% RSLogix 500 project LINL0619_042121 download.RSS, saved by version 11.00.00.00 %
PROJECT "LINL0619"    % processor: MicroLogix 1400 %

PROGRAM FILES
  LAD 2   65 rungs
  LAD 3   9 rungs
  LAD 4   18 rungs
  LAD 5   11 rungs
  LAD 6   13 rungs
  LAD 7   5 rungs
  LAD 8   5 rungs
  LAD 9   26 rungs
  LAD 10   5 rungs
  LAD 11   6 rungs
  LAD 12   3 rungs
  LAD 13   7 rungs
  LAD 14   7 rungs
  LAD 81   21 rungs
  LAD 82   8 rungs
  LAD 83   6 rungs
  LAD 84   4 rungs
  LAD 85   9 rungs
  LAD 86   5 rungs
  LAD 87   5 rungs
  LAD 90   3 rungs
  LAD 91   9 rungs
  LAD 92   5 rungs
  LAD 93   3 rungs
  LAD 94   21 rungs
  LAD 95   7 rungs
  LAD 96   6 rungs
  LAD 97   4 rungs
  LAD 98   8 rungs
  LAD 99   5 rungs
  LAD 100   5 rungs
  LAD 101   7 rungs
  LAD 102   8 rungs
  LAD 103   3 rungs
  LAD 104   9 rungs
  LAD 105   7 rungs
  LAD 106   3 rungs
  LAD 135   3 rungs
  LAD 137   15 rungs
  LAD 138   13 rungs
  LAD 139   19 rungs
  LAD 140   8 rungs
  LAD 141   6 rungs
  LAD 142   6 rungs
  LAD 143   7 rungs
  LAD 144   8 rungs
  LAD 148   21 rungs
  LAD 149   7 rungs
  LAD 150   6 rungs
  LAD 151   4 rungs
  LAD 152   9 rungs
  LAD 153   5 rungs
  LAD 154   5 rungs
  LAD 155   10 rungs
  LAD 156   8 rungs
  LAD 157   3 rungs
  LAD 158   9 rungs
  LAD 159   5 rungs
  LAD 160   3 rungs
  LAD 161   21 rungs
  LAD 162   7 rungs
  LAD 163   5 rungs
  LAD 164   3 rungs
  LAD 165   8 rungs
  LAD 166   5 rungs
  LAD 167   5 rungs
  LAD 168   9 rungs
  LAD 169   8 rungs
  LAD 170   3 rungs
  LAD 171   9 rungs
  LAD 172   5 rungs
  LAD 173   3 rungs
  LAD 174   22 rungs
  LAD 175   7 rungs
  LAD 176   6 rungs
  LAD 177   4 rungs
  LAD 178   9 rungs
  LAD 179   5 rungs
  LAD 180   5 rungs
  LAD 181   9 rungs
  LAD 182   8 rungs
  LAD 183   3 rungs
  LAD 184   9 rungs
  LAD 185   5 rungs
  LAD 186   3 rungs
  LAD 187   22 rungs
  LAD 188   7 rungs
  LAD 189   6 rungs
  LAD 190   4 rungs
  LAD 191   9 rungs
  LAD 192   5 rungs
  LAD 193   5 rungs
  LAD 194   9 rungs
  LAD 195   8 rungs
  LAD 196   3 rungs
  LAD 197   9 rungs
  LAD 198   5 rungs
  LAD 199   3 rungs
  LAD 200   16 rungs
  LAD 235   7 rungs
  LAD 236   5 rungs
  LAD 237   4 rungs
  LAD 238   4 rungs
  LAD 239   4 rungs
  LAD 240   4 rungs
  LAD 241   4 rungs
  LAD 242   4 rungs
  LAD 243   4 rungs
  LAD 244   31 rungs
  LAD 245   8 rungs
  LAD 246   9 rungs
  LAD 247   6 rungs
  LAD 248   6 rungs
  LAD 249   8 rungs
  LAD 250   8 rungs
  LAD 251   8 rungs
  LAD 252   7 rungs
  LAD 253   7 rungs
  LAD 254   4 rungs
  LAD 255   18 rungs
  LAD 88, 89, 107, 108, 109, 110, 111, 112, 113, 114, 115, 116, 117, 118, 119, 120, 121, 122, 123, 124, 125, 126, 127, 128, 129, 130, 131, 132: only END

DATA FILES
  O0 OUTPUT  11 elements
  I1 INPUT  11 elements
  S2 STATUS  66 elements
  B3 BINARY  256 elements
  T4 TIMER  45 elements
  C5 COUNTER  1 elements
  R6 CONTROL  30 elements
  N7 INTEGER  200 elements
  F8 FLOAT  1 elements
  L13   256 elements
  L19   50 elements
  L20   256 elements
  L21   256 elements
  L22   50 elements
  L23   50 elements
  L30   50 elements
  L31   50 elements
  L32   50 elements
  L33   50 elements
  B34   128 elements
  B35   128 elements
  B36   128 elements
  B37   128 elements
  B38   1 elements
  B39   128 elements
  B40   1 elements
  B41   128 elements
  B100   100 elements
  N101   256 elements
  L102   256 elements

LADDER 2
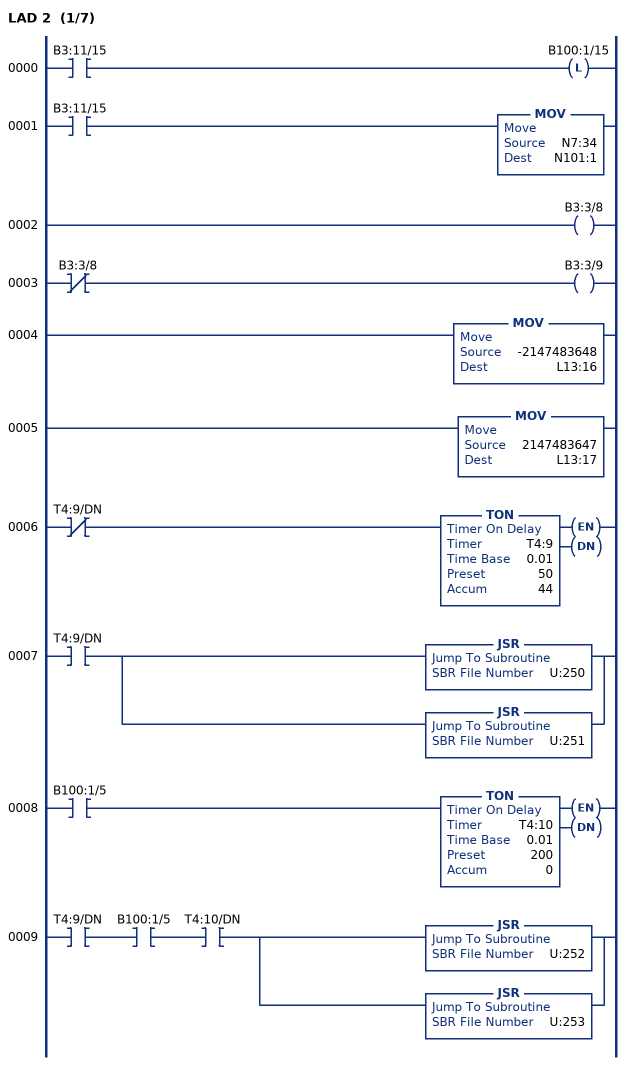
% Rung: 0 %
SOR XIC B3:11/15 OTL B100:1/15 EOR
% Rung: 1 %
SOR XIC B3:11/15 MOV N7:34 N101:1 EOR
% Rung: 2 %
SOR OTE B3:3/8 EOR
% Rung: 3 %
SOR XIO B3:3/8 OTE B3:3/9 EOR
% Rung: 4 %
SOR MOV -2147483648 L13:16 EOR
% Rung: 5 %
SOR MOV 2147483647 L13:17 EOR
% Rung: 6 %
SOR XIO T4:9/DN TON T4:9 0.01 50 44 EOR
% Rung: 7 %
SOR XIC T4:9/DN BST JSR U:250 NXB JSR U:251 BND EOR
% Rung: 8 %
SOR XIC B100:1/5 TON T4:10 0.01 200 0 EOR
% Rung: 9 %
SOR XIC T4:9/DN XIC B100:1/5 XIC T4:10/DN BST JSR U:252 NXB JSR U:253 BND EOR

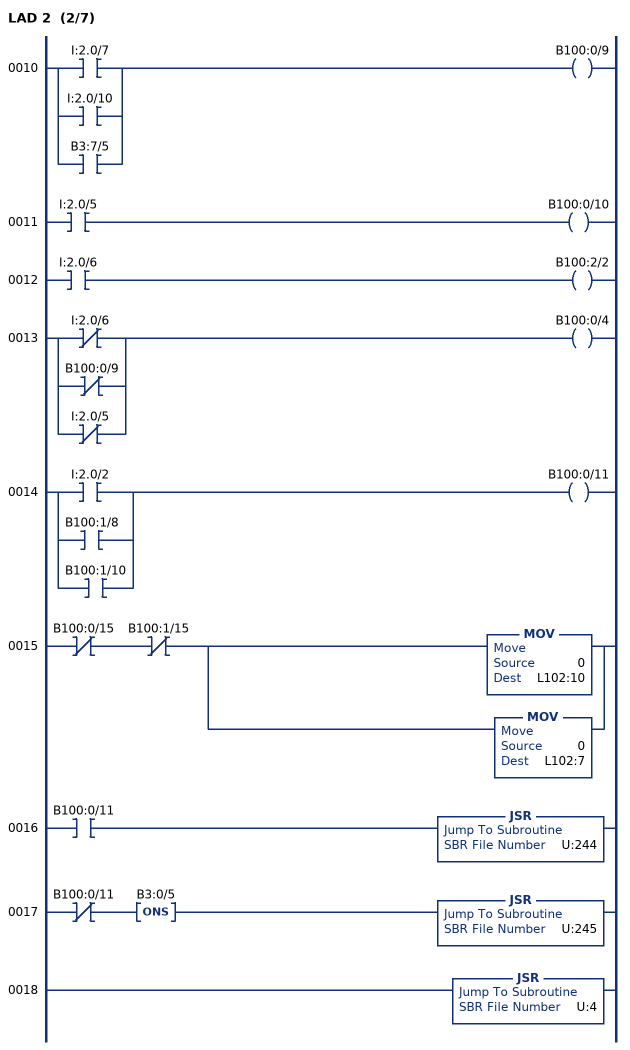
% Rung: 10 %
SOR BST XIC I:2.0/7 NXB XIC I:2.0/10 NXB XIC B3:7/5 BND OTE B100:0/9 EOR
% Rung: 11 %
SOR XIC I:2.0/5 OTE B100:0/10 EOR
% Rung: 12 %
SOR XIC I:2.0/6 OTE B100:2/2 EOR
% Rung: 13 %
SOR BST XIO I:2.0/6 NXB XIO B100:0/9 NXB XIO I:2.0/5 BND OTE B100:0/4 EOR
% Rung: 14 %
SOR BST XIC I:2.0/2 NXB XIC B100:1/8 NXB XIC B100:1/10 BND OTE B100:0/11 EOR
% Rung: 15 %
SOR XIO B100:0/15 XIO B100:1/15 BST MOV 0 L102:10 NXB MOV 0 L102:7 BND EOR
% Rung: 16 %
SOR XIC B100:0/11 JSR U:244 EOR
% Rung: 17 %
SOR XIO B100:0/11 ONS B3:0/5 JSR U:245 EOR
% Rung: 18 %
SOR JSR U:4 EOR

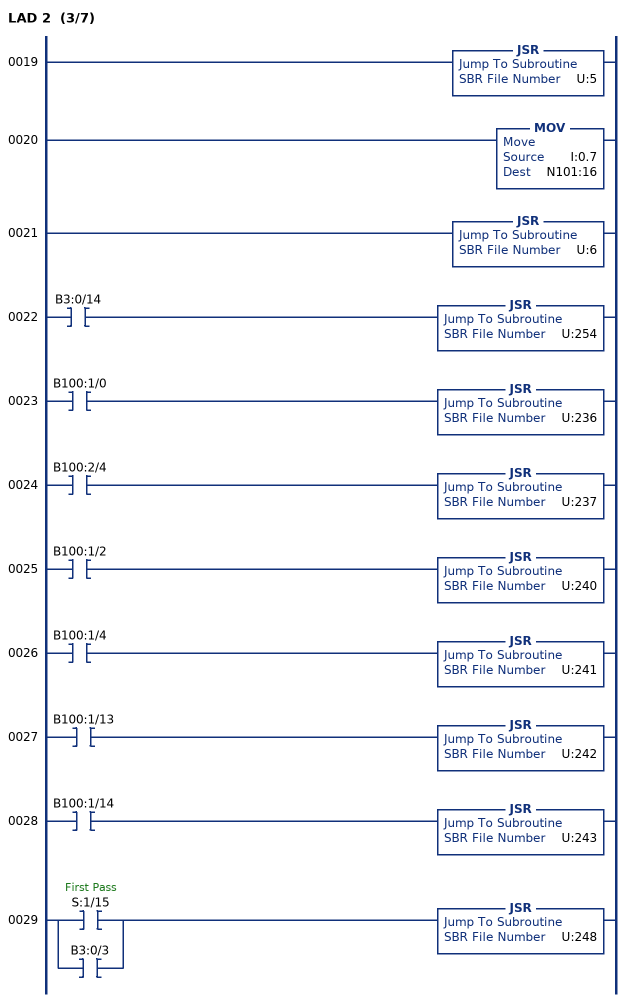
% Rung: 19 %
SOR JSR U:5 EOR
% Rung: 20 %
SOR MOV I:0.7 N101:16 EOR
% Rung: 21 %
SOR JSR U:6 EOR
% Rung: 22 %
SOR XIC B3:0/14 JSR U:254 EOR
% Rung: 23 %
SOR XIC B100:1/0 JSR U:236 EOR
% Rung: 24 %
SOR XIC B100:2/4 JSR U:237 EOR
% Rung: 25 %
SOR XIC B100:1/2 JSR U:240 EOR
% Rung: 26 %
SOR XIC B100:1/4 JSR U:241 EOR
% Rung: 27 %
SOR XIC B100:1/13 JSR U:242 EOR
% Rung: 28 %
SOR XIC B100:1/14 JSR U:243 EOR
% Rung: 29 %
SOR BST XIC S:1/15 NXB XIC B3:0/3 BND JSR U:248 EOR
%   S:1/15  "First Pass" %

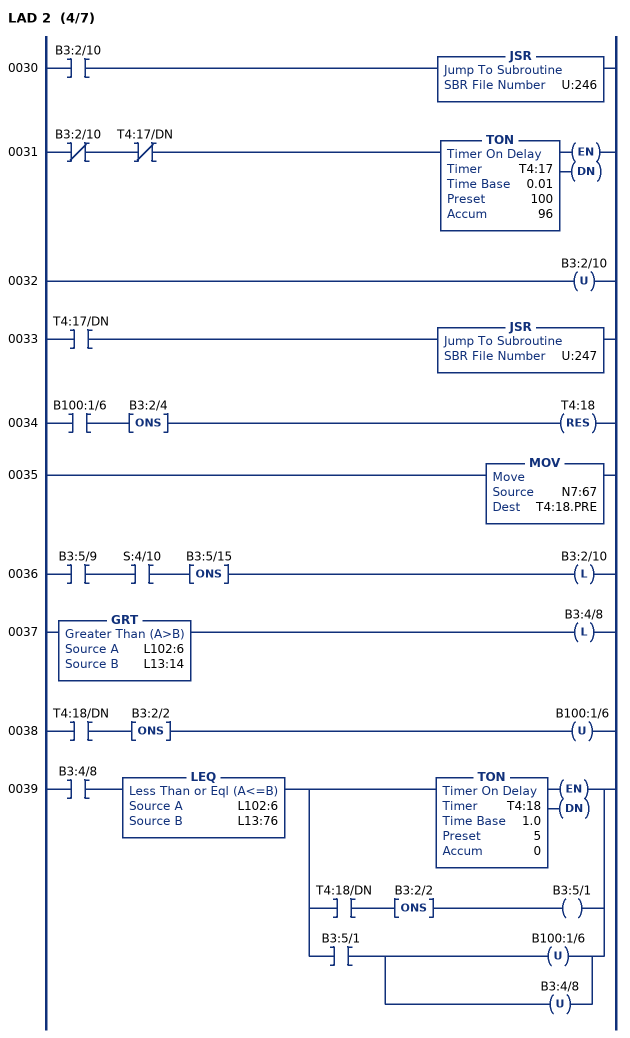
% Rung: 30 %
SOR XIC B3:2/10 JSR U:246 EOR
% Rung: 31 %
SOR XIO B3:2/10 XIO T4:17/DN TON T4:17 0.01 100 96 EOR
% Rung: 32 %
SOR OTU B3:2/10 EOR
% Rung: 33 %
SOR XIC T4:17/DN JSR U:247 EOR
% Rung: 34 %
SOR XIC B100:1/6 ONS B3:2/4 RES T4:18 EOR
% Rung: 35 %
SOR MOV N7:67 T4:18.PRE EOR
% Rung: 36 %
SOR XIC B3:5/9 XIC S:4/10 ONS B3:5/15 OTL B3:2/10 EOR
% Rung: 37 %
SOR GRT L102:6 L13:14 OTL B3:4/8 EOR
% Rung: 38 %
SOR XIC T4:18/DN ONS B3:2/2 OTU B100:1/6 EOR
% Rung: 39 %
SOR XIC B3:4/8 LEQ L102:6 L13:76 BST TON T4:18 1.0 5 0 NXB XIC T4:18/DN ONS B3:2/2 OTE B3:5/1 NXB XIC B3:5/1 BST OTU B100:1/6 NXB OTU B3:4/8 BND BND EOR

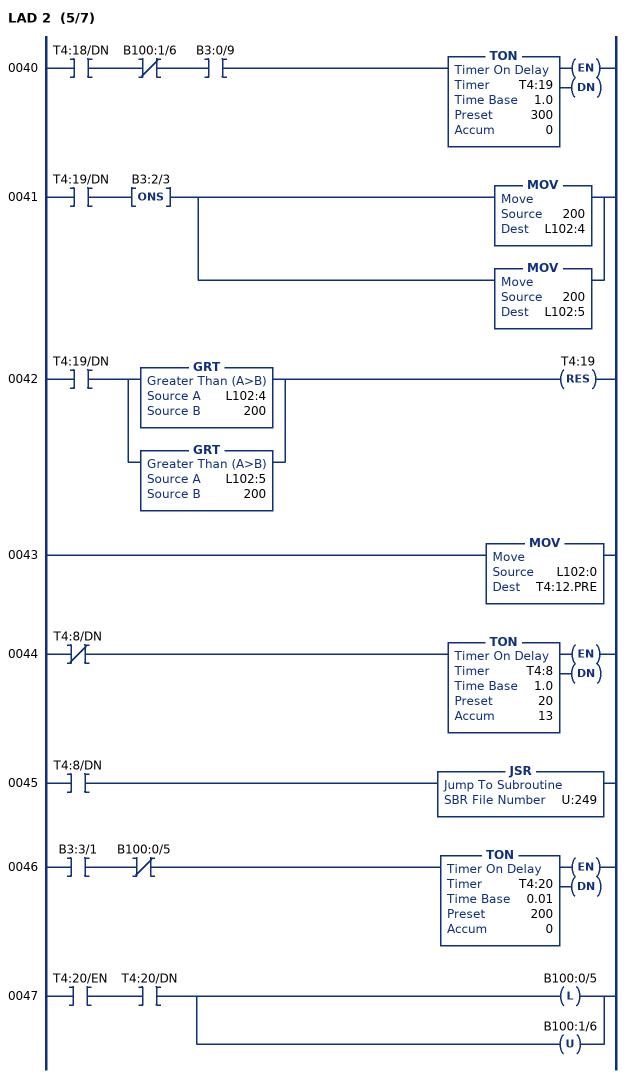
% Rung: 40 %
SOR XIC T4:18/DN XIO B100:1/6 XIC B3:0/9 TON T4:19 1.0 300 0 EOR
% Rung: 41 %
SOR XIC T4:19/DN ONS B3:2/3 BST MOV 200 L102:4 NXB MOV 200 L102:5 BND EOR
% Rung: 42 %
SOR XIC T4:19/DN BST GRT L102:4 200 NXB GRT L102:5 200 BND RES T4:19 EOR
% Rung: 43 %
SOR MOV L102:0 T4:12.PRE EOR
% Rung: 44 %
SOR XIO T4:8/DN TON T4:8 1.0 20 13 EOR
% Rung: 45 %
SOR XIC T4:8/DN JSR U:249 EOR
% Rung: 46 %
SOR XIC B3:3/1 XIO B100:0/5 TON T4:20 0.01 200 0 EOR
% Rung: 47 %
SOR XIC T4:20/EN XIC T4:20/DN BST OTL B100:0/5 NXB OTU B100:1/6 BND EOR

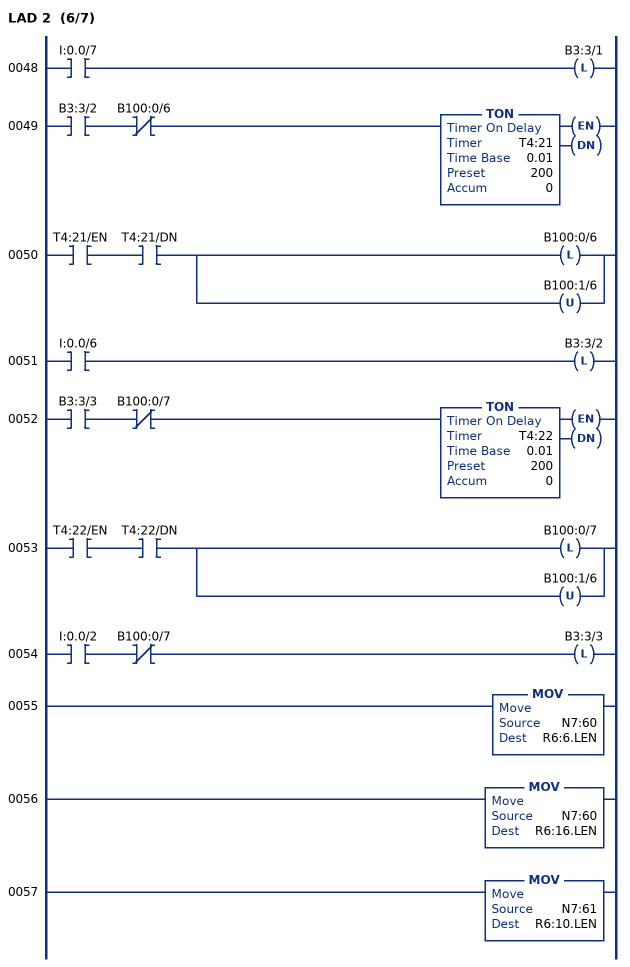
% Rung: 48 %
SOR XIC I:0.0/7 OTL B3:3/1 EOR
% Rung: 49 %
SOR XIC B3:3/2 XIO B100:0/6 TON T4:21 0.01 200 0 EOR
% Rung: 50 %
SOR XIC T4:21/EN XIC T4:21/DN BST OTL B100:0/6 NXB OTU B100:1/6 BND EOR
% Rung: 51 %
SOR XIC I:0.0/6 OTL B3:3/2 EOR
% Rung: 52 %
SOR XIC B3:3/3 XIO B100:0/7 TON T4:22 0.01 200 0 EOR
% Rung: 53 %
SOR XIC T4:22/EN XIC T4:22/DN BST OTL B100:0/7 NXB OTU B100:1/6 BND EOR
% Rung: 54 %
SOR XIC I:0.0/2 XIO B100:0/7 OTL B3:3/3 EOR
% Rung: 55 %
SOR MOV N7:60 R6:6.LEN EOR
% Rung: 56 %
SOR MOV N7:60 R6:16.LEN EOR
% Rung: 57 %
SOR MOV N7:61 R6:10.LEN EOR

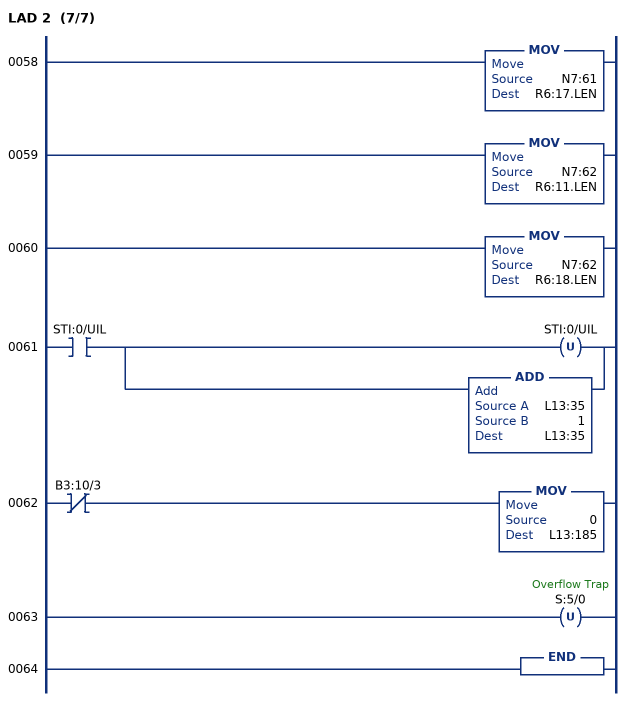
% Rung: 58 %
SOR MOV N7:61 R6:17.LEN EOR
% Rung: 59 %
SOR MOV N7:62 R6:11.LEN EOR
% Rung: 60 %
SOR MOV N7:62 R6:18.LEN EOR
% Rung: 61 %
SOR XIC STI:0/UIL BST OTU STI:0/UIL NXB ADD L13:35 1 L13:35 BND EOR
% Rung: 62 %
SOR XIO B3:10/3 MOV 0 L13:185 EOR
% Rung: 63 %
SOR OTU S:5/0 EOR
%   S:5/0  "Overflow Trap" %
% Rung: 64 %
SOR END EOR

LADDER 3
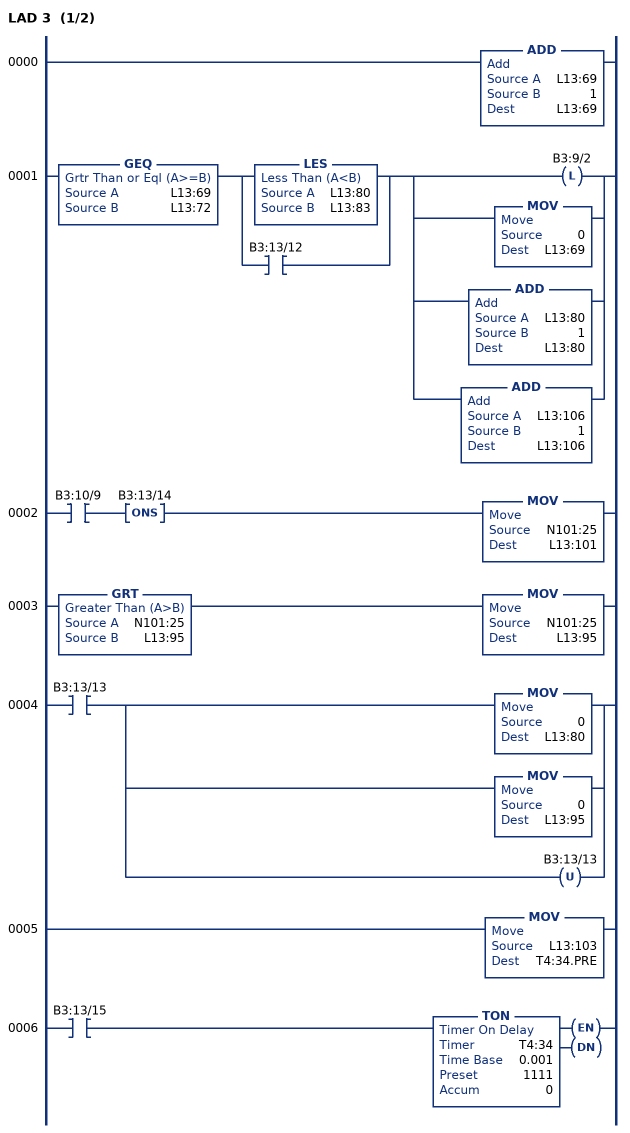
% Rung: 0 %
SOR ADD L13:69 1 L13:69 EOR
% Rung: 1 %
SOR GEQ L13:69 L13:72 BST LES L13:80 L13:83 NXB XIC B3:13/12 BND BST OTL B3:9/2 NXB MOV 0 L13:69 NXB ADD L13:80 1 L13:80 NXB ADD L13:106 1 L13:106 BND EOR
% Rung: 2 %
SOR XIC B3:10/9 ONS B3:13/14 MOV N101:25 L13:101 EOR
% Rung: 3 %
SOR GRT N101:25 L13:95 MOV N101:25 L13:95 EOR
% Rung: 4 %
SOR XIC B3:13/13 BST MOV 0 L13:80 NXB MOV 0 L13:95 NXB OTU B3:13/13 BND EOR
% Rung: 5 %
SOR MOV L13:103 T4:34.PRE EOR
% Rung: 6 %
SOR XIC B3:13/15 TON T4:34 0.001 1111 0 EOR

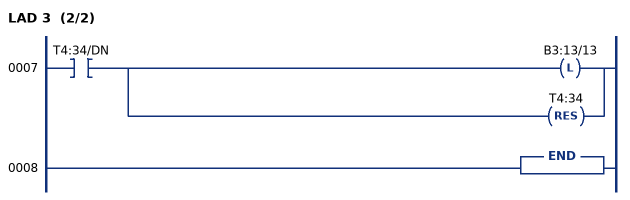
% Rung: 7 %
SOR XIC T4:34/DN BST OTL B3:13/13 NXB RES T4:34 BND EOR
% Rung: 8 %
SOR END EOR

LADDER 4
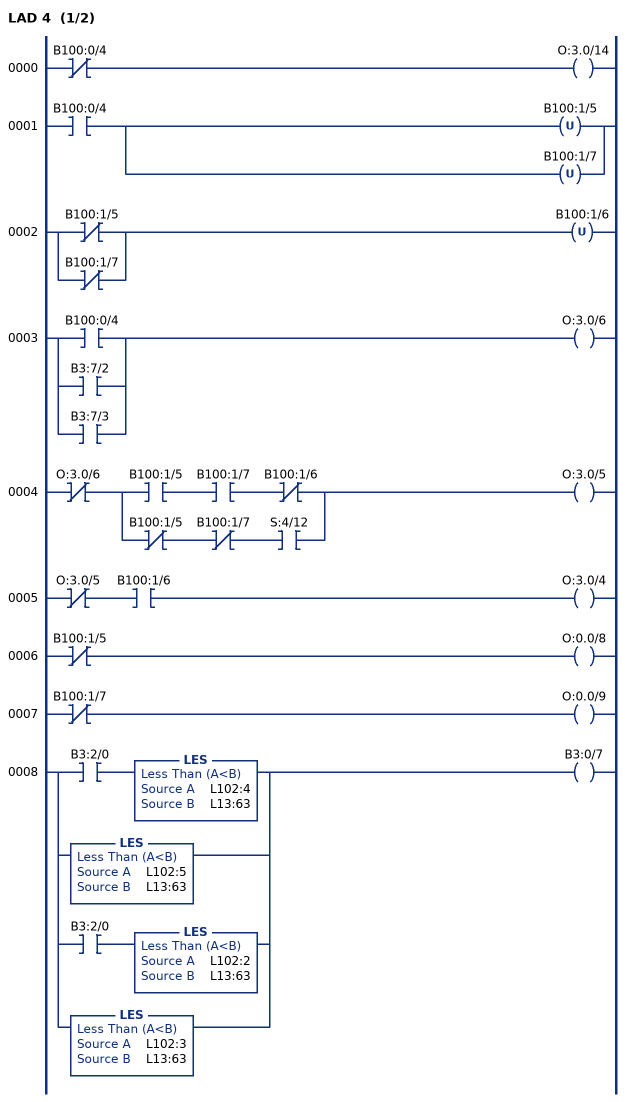
% Rung: 0 %
SOR XIO B100:0/4 OTE O:3.0/14 EOR
% Rung: 1 %
SOR XIC B100:0/4 BST OTU B100:1/5 NXB OTU B100:1/7 BND EOR
% Rung: 2 %
SOR BST XIO B100:1/5 NXB XIO B100:1/7 BND OTU B100:1/6 EOR
% Rung: 3 %
SOR BST XIC B100:0/4 NXB XIC B3:7/2 NXB XIC B3:7/3 BND OTE O:3.0/6 EOR
% Rung: 4 %
SOR XIO O:3.0/6 BST XIC B100:1/5 XIC B100:1/7 XIO B100:1/6 NXB XIO B100:1/5 XIO B100:1/7 XIC S:4/12 BND OTE O:3.0/5 EOR
% Rung: 5 %
SOR XIO O:3.0/5 XIC B100:1/6 OTE O:3.0/4 EOR
% Rung: 6 %
SOR XIO B100:1/5 OTE O:0.0/8 EOR
% Rung: 7 %
SOR XIO B100:1/7 OTE O:0.0/9 EOR
% Rung: 8 %
SOR BST XIC B3:2/0 LES L102:4 L13:63 NXB LES L102:5 L13:63 NXB XIC B3:2/0 LES L102:2 L13:63 NXB LES L102:3 L13:63 BND OTE B3:0/7 EOR

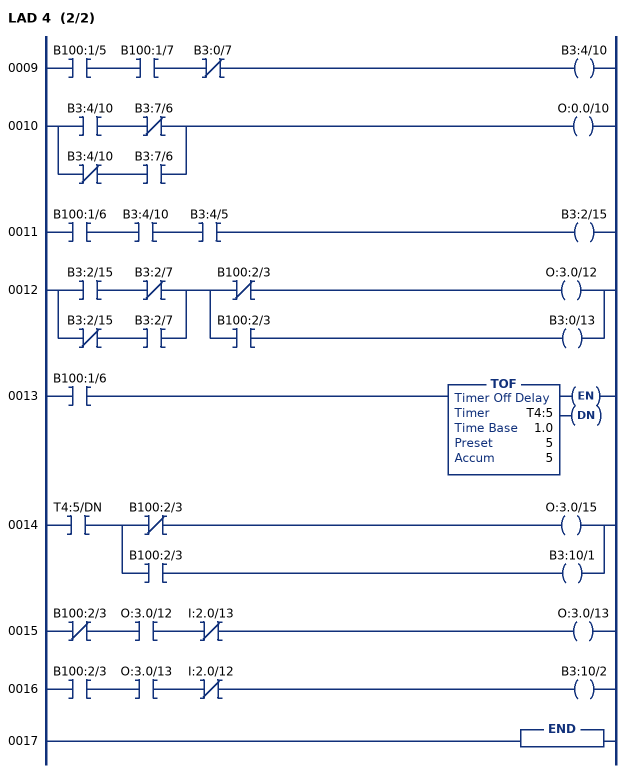
% Rung: 9 %
SOR XIC B100:1/5 XIC B100:1/7 XIO B3:0/7 OTE B3:4/10 EOR
% Rung: 10 %
SOR BST XIC B3:4/10 XIO B3:7/6 NXB XIO B3:4/10 XIC B3:7/6 BND OTE O:0.0/10 EOR
% Rung: 11 %
SOR XIC B100:1/6 XIC B3:4/10 XIC B3:4/5 OTE B3:2/15 EOR
% Rung: 12 %
SOR BST XIC B3:2/15 XIO B3:2/7 NXB XIO B3:2/15 XIC B3:2/7 BND BST XIO B100:2/3 OTE O:3.0/12 NXB XIC B100:2/3 OTE B3:0/13 BND EOR
% Rung: 13 %
SOR XIC B100:1/6 TOF T4:5 1.0 5 5 EOR
% Rung: 14 %
SOR XIC T4:5/DN BST XIO B100:2/3 OTE O:3.0/15 NXB XIC B100:2/3 OTE B3:10/1 BND EOR
% Rung: 15 %
SOR XIO B100:2/3 XIC O:3.0/12 XIO I:2.0/13 OTE O:3.0/13 EOR
% Rung: 16 %
SOR XIC B100:2/3 XIC O:3.0/13 XIO I:2.0/12 OTE B3:10/2 EOR
% Rung: 17 %
SOR END EOR

LADDER 5
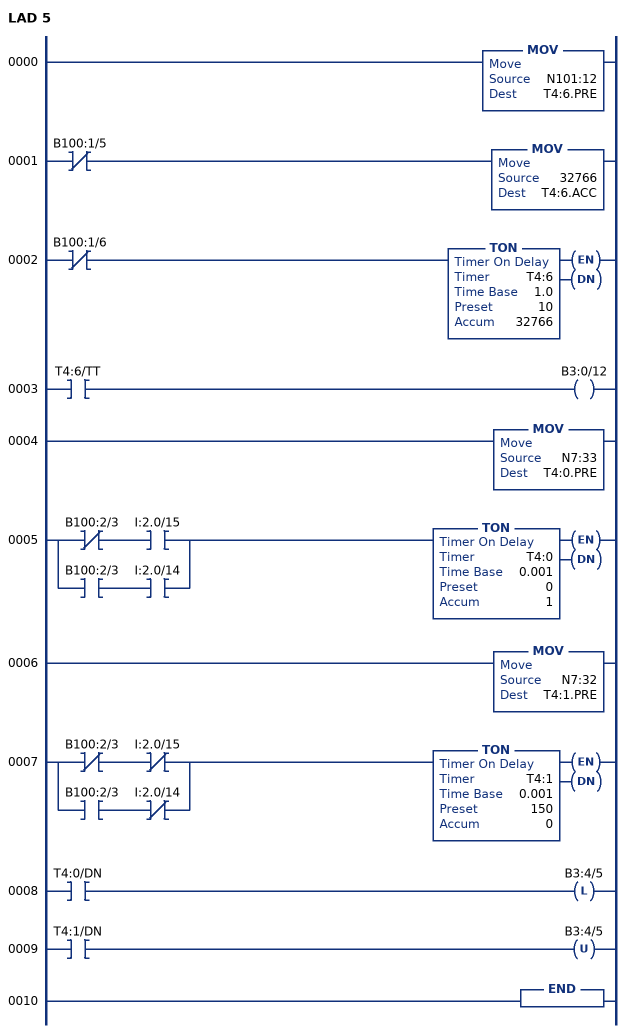
% Rung: 0 %
SOR MOV N101:12 T4:6.PRE EOR
% Rung: 1 %
SOR XIO B100:1/5 MOV 32766 T4:6.ACC EOR
% Rung: 2 %
SOR XIO B100:1/6 TON T4:6 1.0 10 32766 EOR
% Rung: 3 %
SOR XIC T4:6/TT OTE B3:0/12 EOR
% Rung: 4 %
SOR MOV N7:33 T4:0.PRE EOR
% Rung: 5 %
SOR BST XIO B100:2/3 XIC I:2.0/15 NXB XIC B100:2/3 XIC I:2.0/14 BND TON T4:0 0.001 0 1 EOR
% Rung: 6 %
SOR MOV N7:32 T4:1.PRE EOR
% Rung: 7 %
SOR BST XIO B100:2/3 XIO I:2.0/15 NXB XIC B100:2/3 XIO I:2.0/14 BND TON T4:1 0.001 150 0 EOR
% Rung: 8 %
SOR XIC T4:0/DN OTL B3:4/5 EOR
% Rung: 9 %
SOR XIC T4:1/DN OTU B3:4/5 EOR
% Rung: 10 %
SOR END EOR

LADDER 6
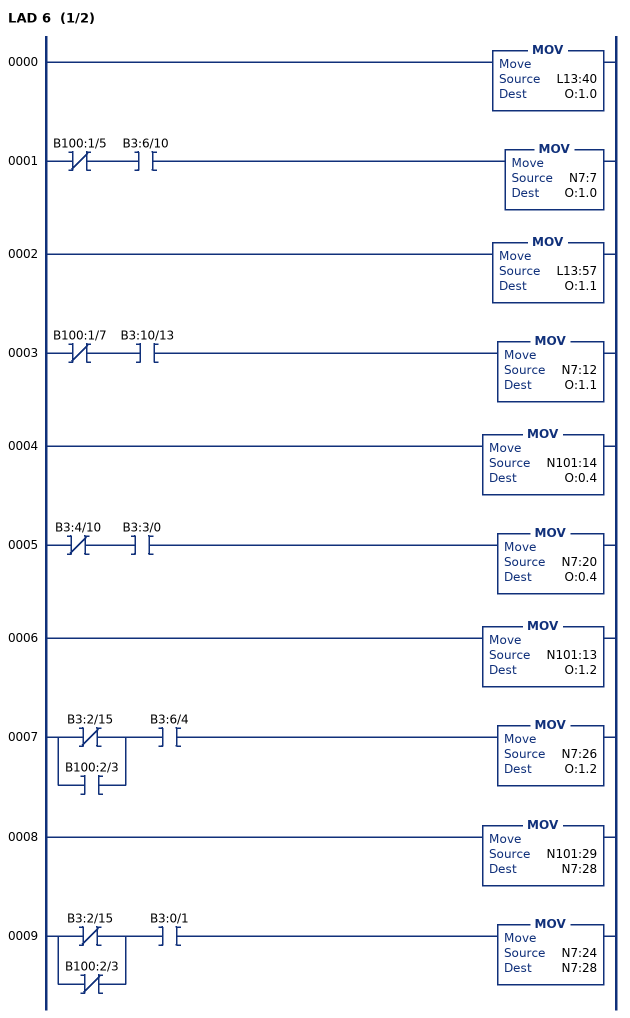
% Rung: 0 %
SOR MOV L13:40 O:1.0 EOR
% Rung: 1 %
SOR XIO B100:1/5 XIC B3:6/10 MOV N7:7 O:1.0 EOR
% Rung: 2 %
SOR MOV L13:57 O:1.1 EOR
% Rung: 3 %
SOR XIO B100:1/7 XIC B3:10/13 MOV N7:12 O:1.1 EOR
% Rung: 4 %
SOR MOV N101:14 O:0.4 EOR
% Rung: 5 %
SOR XIO B3:4/10 XIC B3:3/0 MOV N7:20 O:0.4 EOR
% Rung: 6 %
SOR MOV N101:13 O:1.2 EOR
% Rung: 7 %
SOR BST XIO B3:2/15 NXB XIC B100:2/3 BND XIC B3:6/4 MOV N7:26 O:1.2 EOR
% Rung: 8 %
SOR MOV N101:29 N7:28 EOR
% Rung: 9 %
SOR BST XIO B3:2/15 NXB XIO B100:2/3 BND XIC B3:0/1 MOV N7:24 N7:28 EOR

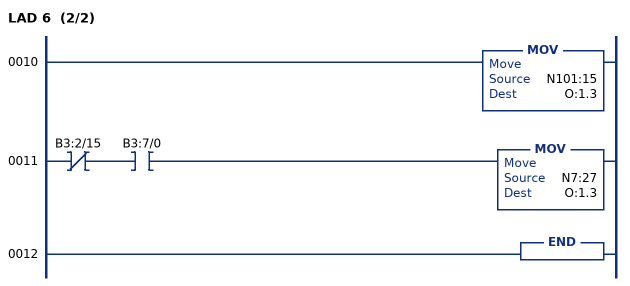
% Rung: 10 %
SOR MOV N101:15 O:1.3 EOR
% Rung: 11 %
SOR XIO B3:2/15 XIC B3:7/0 MOV N7:27 O:1.3 EOR
% Rung: 12 %
SOR END EOR

LADDER 7
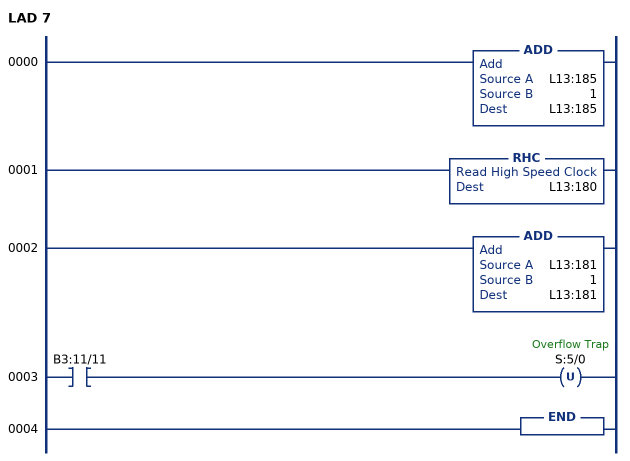
% Rung: 0 %
SOR ADD L13:185 1 L13:185 EOR
% Rung: 1 %
SOR RHC L13:180 EOR
% Rung: 2 %
SOR ADD L13:181 1 L13:181 EOR
% Rung: 3 %
SOR XIC B3:11/11 OTU S:5/0 EOR
%   S:5/0  "Overflow Trap" %
% Rung: 4 %
SOR END EOR

LADDER 8
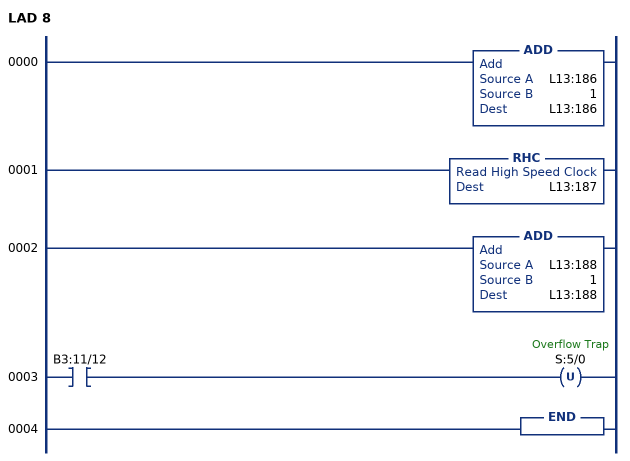
% Rung: 0 %
SOR ADD L13:186 1 L13:186 EOR
% Rung: 1 %
SOR RHC L13:187 EOR
% Rung: 2 %
SOR ADD L13:188 1 L13:188 EOR
% Rung: 3 %
SOR XIC B3:11/12 OTU S:5/0 EOR
%   S:5/0  "Overflow Trap" %
% Rung: 4 %
SOR END EOR

LADDER 9
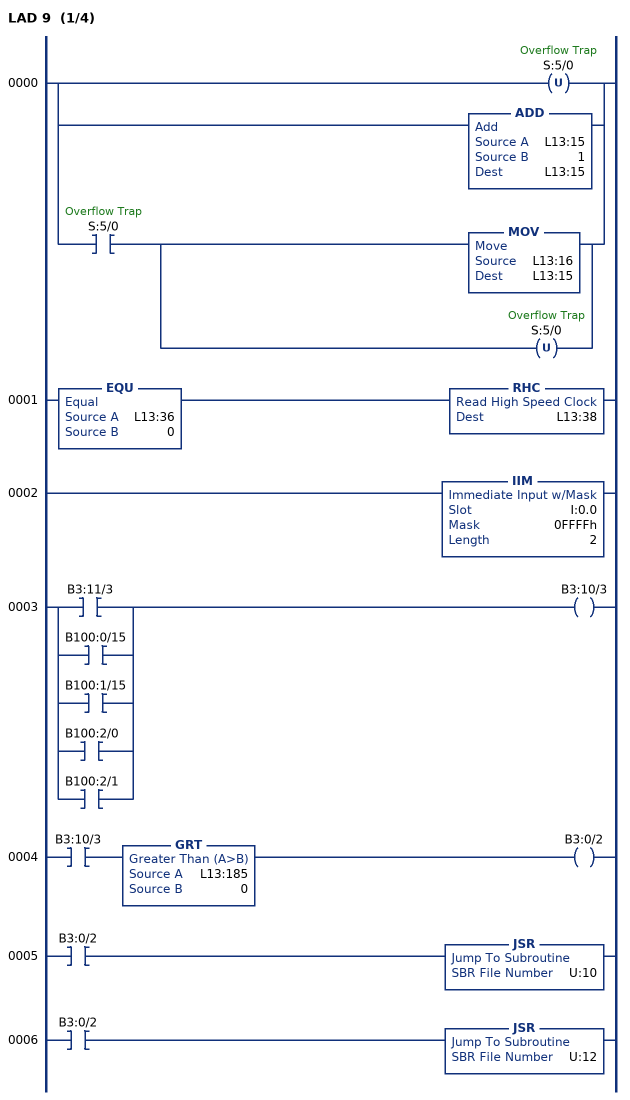
% Rung: 0 %
SOR BST OTU S:5/0 NXB ADD L13:15 1 L13:15 NXB XIC S:5/0 BST MOV L13:16 L13:15 NXB OTU S:5/0 BND BND EOR
%   S:5/0  "Overflow Trap" %
% Rung: 1 %
SOR EQU L13:36 0 RHC L13:38 EOR
% Rung: 2 %
SOR IIM I:0.0 0FFFFh 2 EOR
% Rung: 3 %
SOR BST XIC B3:11/3 NXB XIC B100:0/15 NXB XIC B100:1/15 NXB XIC B100:2/0 NXB XIC B100:2/1 BND OTE B3:10/3 EOR
% Rung: 4 %
SOR XIC B3:10/3 GRT L13:185 0 OTE B3:0/2 EOR
% Rung: 5 %
SOR XIC B3:0/2 JSR U:10 EOR
% Rung: 6 %
SOR XIC B3:0/2 JSR U:12 EOR

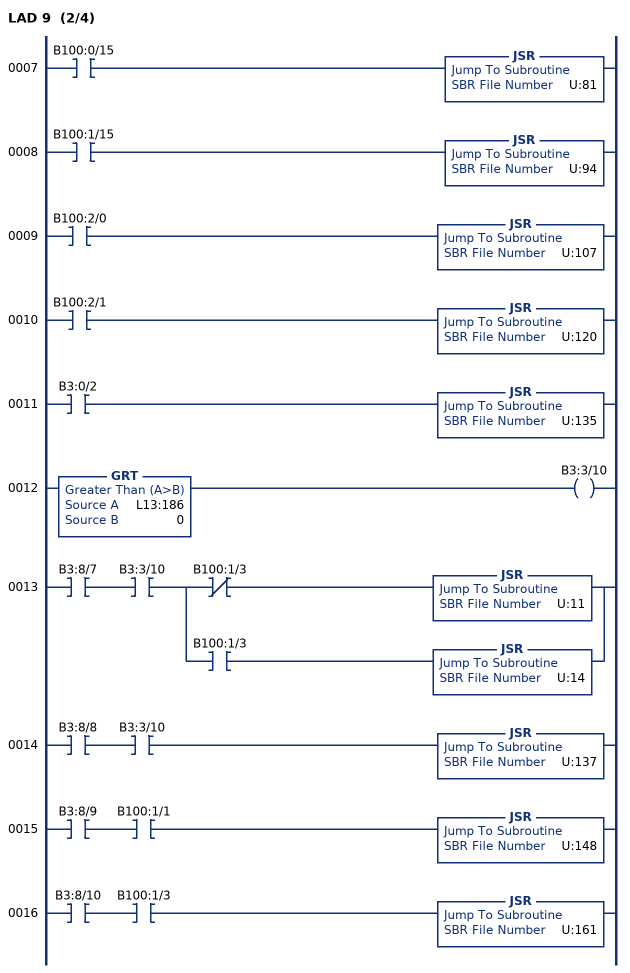
% Rung: 7 %
SOR XIC B100:0/15 JSR U:81 EOR
% Rung: 8 %
SOR XIC B100:1/15 JSR U:94 EOR
% Rung: 9 %
SOR XIC B100:2/0 JSR U:107 EOR
% Rung: 10 %
SOR XIC B100:2/1 JSR U:120 EOR
% Rung: 11 %
SOR XIC B3:0/2 JSR U:135 EOR
% Rung: 12 %
SOR GRT L13:186 0 OTE B3:3/10 EOR
% Rung: 13 %
SOR XIC B3:8/7 XIC B3:3/10 BST XIO B100:1/3 JSR U:11 NXB XIC B100:1/3 JSR U:14 BND EOR
% Rung: 14 %
SOR XIC B3:8/8 XIC B3:3/10 JSR U:137 EOR
% Rung: 15 %
SOR XIC B3:8/9 XIC B100:1/1 JSR U:148 EOR
% Rung: 16 %
SOR XIC B3:8/10 XIC B100:1/3 JSR U:161 EOR

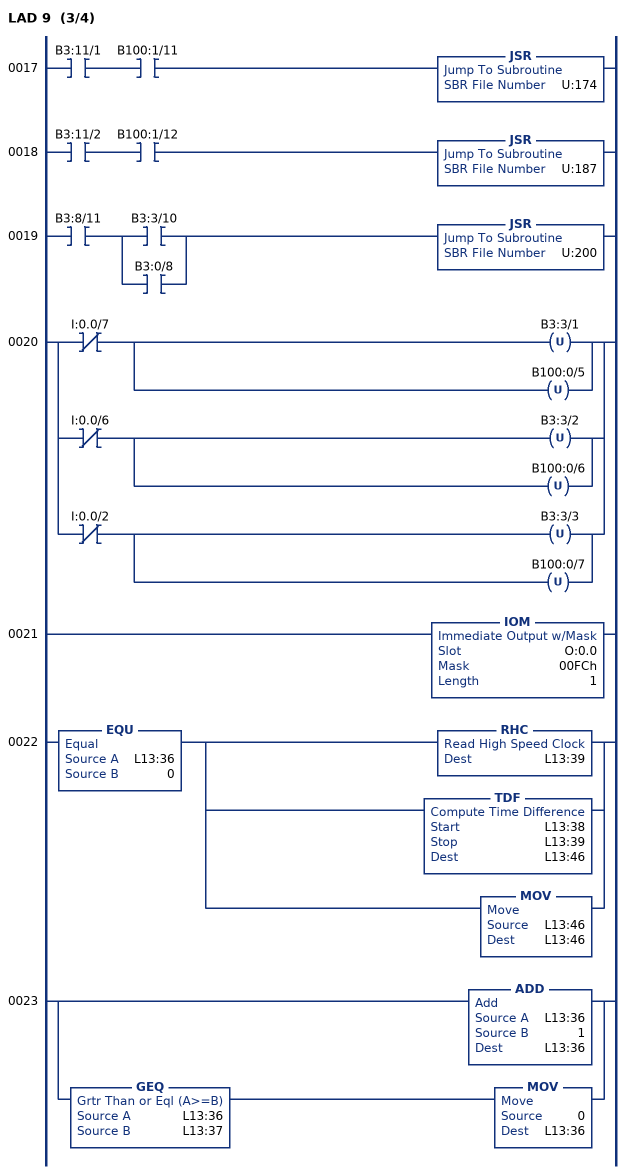
% Rung: 17 %
SOR XIC B3:11/1 XIC B100:1/11 JSR U:174 EOR
% Rung: 18 %
SOR XIC B3:11/2 XIC B100:1/12 JSR U:187 EOR
% Rung: 19 %
SOR XIC B3:8/11 BST XIC B3:3/10 NXB XIC B3:0/8 BND JSR U:200 EOR
% Rung: 20 %
SOR BST XIO I:0.0/7 BST OTU B3:3/1 NXB OTU B100:0/5 BND NXB XIO I:0.0/6 BST OTU B3:3/2 NXB OTU B100:0/6 BND NXB XIO I:0.0/2 BST OTU B3:3/3 NXB OTU B100:0/7 BND BND EOR
% Rung: 21 %
SOR IOM O:0.0 00FCh 1 EOR
% Rung: 22 %
SOR EQU L13:36 0 BST RHC L13:39 NXB TDF L13:38 L13:39 L13:46 NXB MOV L13:46 L13:46 BND EOR
% Rung: 23 %
SOR BST ADD L13:36 1 L13:36 NXB GEQ L13:36 L13:37 MOV 0 L13:36 BND EOR

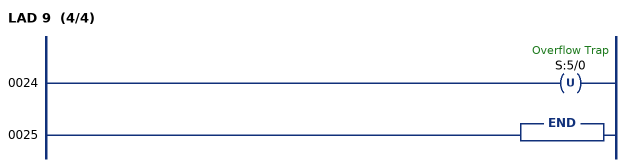
% Rung: 24 %
SOR OTU S:5/0 EOR
%   S:5/0  "Overflow Trap" %
% Rung: 25 %
SOR END EOR

LADDER 10
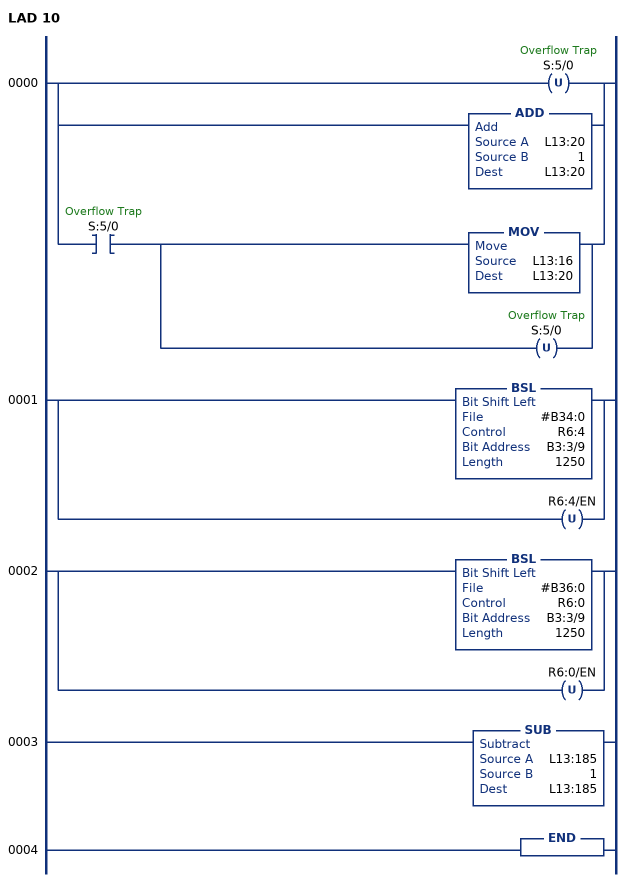
% Rung: 0 %
SOR BST OTU S:5/0 NXB ADD L13:20 1 L13:20 NXB XIC S:5/0 BST MOV L13:16 L13:20 NXB OTU S:5/0 BND BND EOR
%   S:5/0  "Overflow Trap" %
% Rung: 1 %
SOR BST BSL #B34:0 R6:4 B3:3/9 1250 NXB OTU R6:4/EN BND EOR
% Rung: 2 %
SOR BST BSL #B36:0 R6:0 B3:3/9 1250 NXB OTU R6:0/EN BND EOR
% Rung: 3 %
SOR SUB L13:185 1 L13:185 EOR
% Rung: 4 %
SOR END EOR

LADDER 11
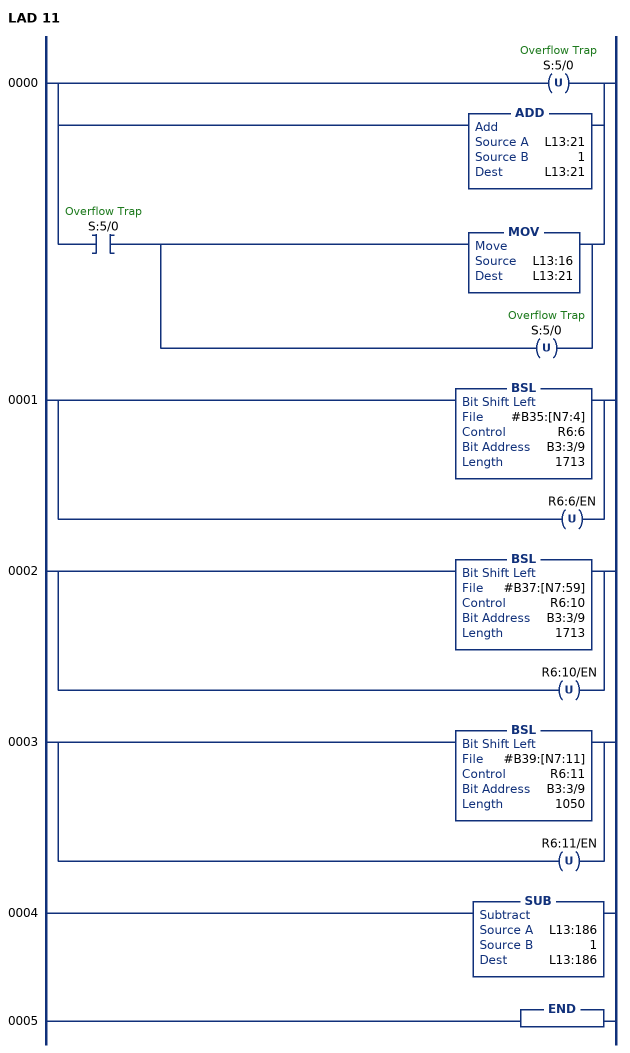
% Rung: 0 %
SOR BST OTU S:5/0 NXB ADD L13:21 1 L13:21 NXB XIC S:5/0 BST MOV L13:16 L13:21 NXB OTU S:5/0 BND BND EOR
%   S:5/0  "Overflow Trap" %
% Rung: 1 %
SOR BST BSL #B35:[N7:4] R6:6 B3:3/9 1713 NXB OTU R6:6/EN BND EOR
% Rung: 2 %
SOR BST BSL #B37:[N7:59] R6:10 B3:3/9 1713 NXB OTU R6:10/EN BND EOR
% Rung: 3 %
SOR BST BSL #B39:[N7:11] R6:11 B3:3/9 1050 NXB OTU R6:11/EN BND EOR
% Rung: 4 %
SOR SUB L13:186 1 L13:186 EOR
% Rung: 5 %
SOR END EOR

LADDER 12
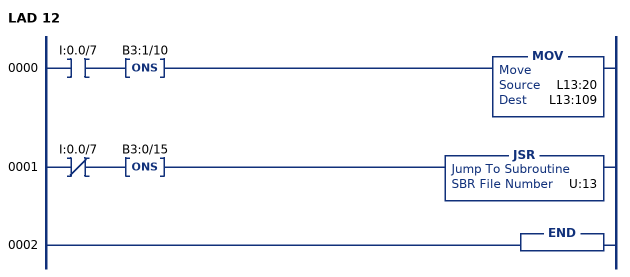
% Rung: 0 %
SOR XIC I:0.0/7 ONS B3:1/10 MOV L13:20 L13:109 EOR
% Rung: 1 %
SOR XIO I:0.0/7 ONS B3:0/15 JSR U:13 EOR
% Rung: 2 %
SOR END EOR

LADDER 13
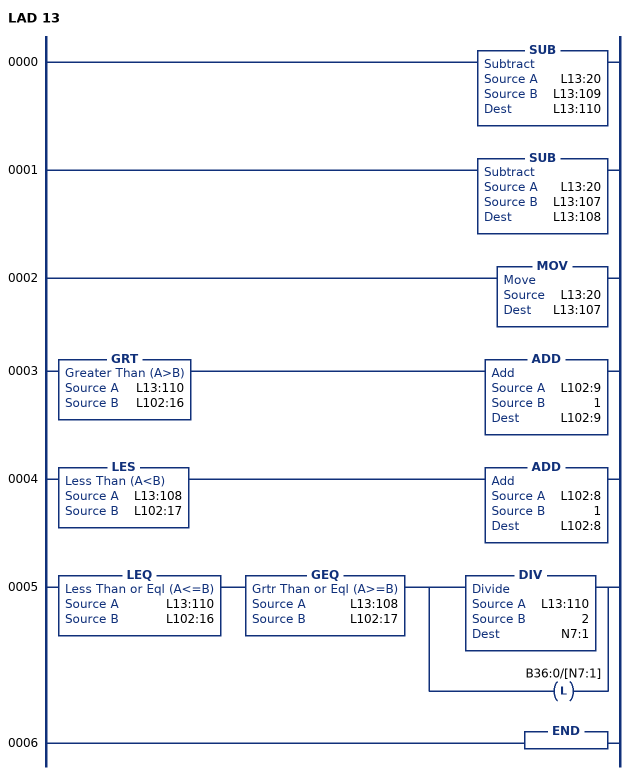
% Rung: 0 %
SOR SUB L13:20 L13:109 L13:110 EOR
% Rung: 1 %
SOR SUB L13:20 L13:107 L13:108 EOR
% Rung: 2 %
SOR MOV L13:20 L13:107 EOR
% Rung: 3 %
SOR GRT L13:110 L102:16 ADD L102:9 1 L102:9 EOR
% Rung: 4 %
SOR LES L13:108 L102:17 ADD L102:8 1 L102:8 EOR
% Rung: 5 %
SOR LEQ L13:110 L102:16 GEQ L13:108 L102:17 BST DIV L13:110 2 N7:1 NXB OTL B36:0/[N7:1] BND EOR
% Rung: 6 %
SOR END EOR

LADDER 14
